INTERFACE I_ResetSequence

METHOD IsReset : BOOL
END_METHOD

END_INTERFACE

(* stored: Version 1.1.0.1
   Itf I_ResetSequence: Id {be808ad5-efdc-4a87-8ed1-6a14424540b4}
   Method IsReset: Id {45dc7d4e-bdb8-4b6d-b313-ba9b6ff84d11} *)
